{attribute 'qualified_only'}
{attribute 'strict'}
{attribute 'to_string'}
TYPE E_ValidationStep :
(
	INITIALIZE := 0,
	WAIT_FOR_IDLE,
	COMMAND_SEQUENCE_START,
	GENERATE_TARGET_POINTS,
	COMMAND_MOVE_TO_FIRST_TARGET,
	COMMAND_START_TRIGGERS,
	CONFIRM_BACK_TO_IDLE
);
END_TYPE

(* stored: Version 1.1.0.1
   DUT E_ValidationStep: Id {22193865-d439-4402-bfa2-d3e98a0a6c40} *)
